// Mitsubishi GX Works2 project: BLOCKRST   PLC: Q03UDV

PROGRAM MAIN
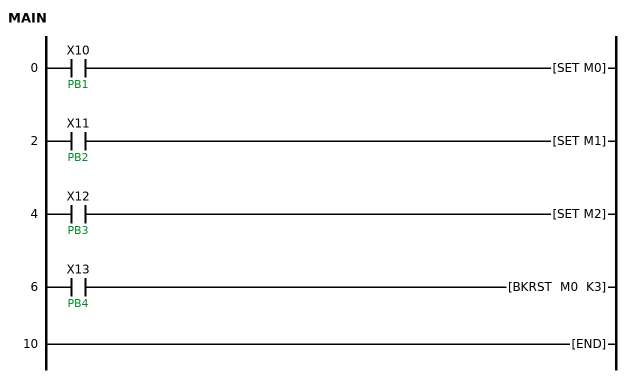
0     LD      X10  ; PB1
      SET     M0
2     LD      X11  ; PB2
      SET     M1
4     LD      X12  ; PB3
      SET     M2
6     LD      X13  ; PB4
      BKRST   M0 K3
10    END
END_PROGRAM
